FUNCTION_BLOCK EL3041
VAR
	_io : EL3xx1_Data;
	{attribute addProperty Name "WcState"}
	_wcState : WcStateInputToggle;
	{attribute addProperty Name "Info data"}
	_infoData : InfoDataAds;
END_VAR

PROPERTY IO : REFERENCE TO EL3xx1_Data
GET
IO REF= _io;
END_GET
END_PROPERTY

PROPERTY WcState : REFERENCE TO WcStateInputToggle
GET
WcState REF= _wcState;
END_GET
END_PROPERTY

END_FUNCTION_BLOCK

(* stored: Version 1.1.0.1, ProductVersion 3.1.4024.9
   POU EL3041: Id {6333ec1b-c393-04d8-375c-ddda9ca9cd23}, SpecialFunc None
   Property IO: Id {f7c10a49-5055-0c69-0fc8-7b63150d573b}
   Get Get: Id {b6eb331f-f8a7-0b94-054f-3b392cebcd80}
   Property WcState: Id {9a7885d1-f7dd-01be-3fe9-91a130ad0a77}
   Get Get: Id {26c5750d-65c3-035a-25e7-30260bf3ed59} *)
